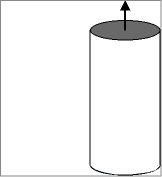
VISUALIZATION VISU_Tube_Top_12  // 162x177
VAR_IN_OUT
	azi : LREAL;
END_VAR
    Ellipse (90,155 70x20)
        p2858320360: azi
    Polygon (90,30) (160,30) (160,165) (155,170) (148,172) (140,173) (132,174) (122,174) (114,174) (104,172) (95,169) (90,165)
        p2858320360: azi
    Ellipse (90,20 70x20)
        p2858320360: azi
    Polygon (120,10) (125,0) (130,10)
        p2858320360: azi
    Polyline (125,30) (125,10)
        p2858320360: azi
    Polyline (90,165) (90,30)
        p2858320360: azi
    Polyline (160,165) (160,30)
        p2858320360: azi
END_VISUALIZATION

(* stored: Version 1.1.0.1, ProductVersion 3.1.4018.5
   Visu VISU_Tube_Top_12: Id {b079ece6-8da3-4366-a364-75a8de26bbda} *)
